FUNCTION_BLOCK TcaSingleAxis EXTENDS TcoDrivesBeckhoff.TcoSingleAxis

VAR
END_VAR

END_FUNCTION_BLOCK

(* stored: Version 1.1.0.1
   POU TcaSingleAxis: Id {96c98aa5-c6ee-4857-a717-4d67b877ad0d}, SpecialFunc None *)
